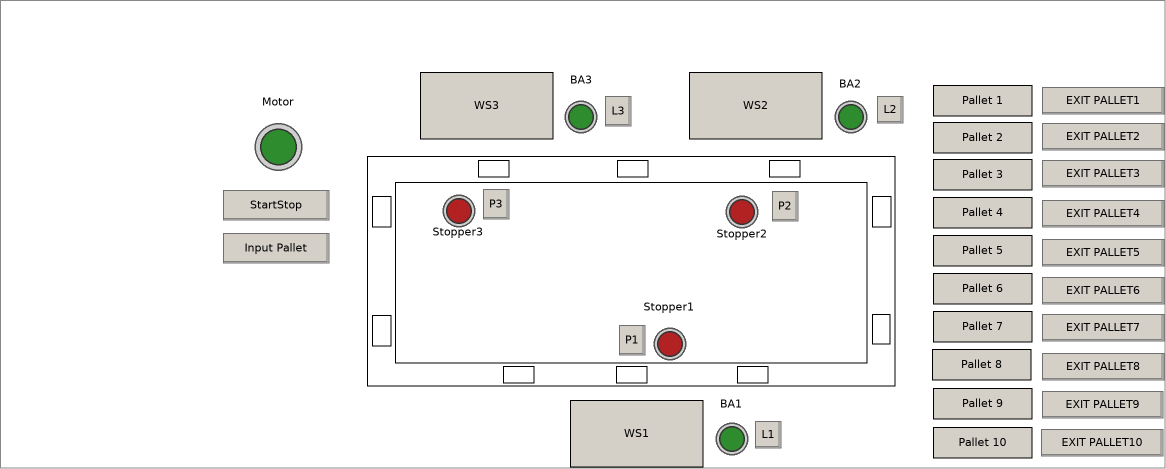
VISUALIZATION Visualization  // 1166x469
    RoundedRectangle (367,156 528x230)
    RoundedRectangle (395,182 472x181)
    Rectangle (570,400 133x67), "WS1", colour toggle: MAIN.T1.Q
    Rectangle (420,72 133x67), "WS3", colour toggle: MAIN.T3.Q
    Rectangle (689,72 133x67), "WS2", colour toggle: MAIN.T2.Q
    Button (755,421 26x27), "L1", text variable: MAIN.L1, colour toggle: MAIN.L1
        toggle MAIN.L1
    Button (605,96 26x30), "L3", text variable: MAIN.L3, colour toggle: MAIN.L3
        toggle MAIN.L3
    Button (483,189 26x30), "P3"
        tap MAIN.P3
    Button (772,191 26x30), "P2"
        tap MAIN.P2
    Button (619,325 26x30), "P1"
        tap MAIN.P1
    Lamp1 (832,94 38x46), tooltip "BA2", variable: MAIN.BA2, style: Lamp-Lamp1-Green
    Label (775,69 150x30), "BA2"
    Lamp1 (562,94 38x46), variable: MAIN.BA3, style: Lamp-Lamp1-Green
    Lamp1 (713,416 38x46), variable: MAIN.BA1, style: Lamp-Lamp1-Green
    Label (506,63 150x34), "BA3"
    Label (656,389 150x30), "BA1"
    Lamp1 (723,189 38x46), variable: MAIN.S2, style: Lamp-Lamp1-Red
    Lamp1 (440,188 38x46), variable: MAIN.S3, style: Lamp-Lamp1-Red
    Lamp1 (651,321 38x46), variable: MAIN.S1, style: Lamp-Lamp1-Red
    Label (594,292 150x30), "Stopper1"
    Label (383,217 150x30), "Stopper3"
    Label (667,219 150x30), "Stopper2"
    Rectangle (503,366 31x17)
    Lamp1 (251,115 55x64), variable: MAIN.MOTOR, style: Lamp-Lamp1-Green
    Label (203,87 150x30), "Motor"
    Button (223,190 106x30), "StartStop"
        toggle MAIN.StartStop
    Button (223,233 106x30), "Input Pallet"
        tap MAIN.INPUT_PALLET_Pressed
    Button (877,96 26x27), "L2", text variable: MAIN.L2, colour toggle: MAIN.L2
        toggle MAIN.L2
    Rectangle (933,85 99x31), "Pallet 1", colour toggle: MAIN.PALLETV[2].WS1
    Rectangle (372,315 19x31)
    Rectangle (617,160 31x17)
    Rectangle (769,160 31x17), invisible if: MAIN.L2
    Rectangle (478,160 31x17), invisible if: MAIN.L3
    Rectangle (737,366 31x17)
    Rectangle (616,366 31x17), invisible if: MAIN.L1
    Rectangle (872,314 18x30)
    Rectangle (872,196 19x31)
    Rectangle (372,196 19x31)
    Rectangle (933,122 99x31), "Pallet 2", colour toggle: MAIN.PALLETV[3].WS1
    Rectangle (933,159 99x31), "Pallet 3", colour toggle: MAIN.PALLETV[4].WS1
    Rectangle (933,197 99x31), "Pallet 4", colour toggle: MAIN.PALLETV[5].WS1
    Rectangle (933,235 99x31), "Pallet 5", colour toggle: MAIN.PALLETV[6].WS1
    Rectangle (933,273 99x31), "Pallet 6", colour toggle: MAIN.PALLETV[7].WS1
    Rectangle (933,311 99x31), "Pallet 7", colour toggle: MAIN.PALLETV[8].WS1
    Rectangle (932,349 99x31), "Pallet 8", colour toggle: MAIN.PALLETV[9].WS1
    Rectangle (933,388 99x31), "Pallet 9", colour toggle: MAIN.PALLETV[10].WS1
    Rectangle (933,427 99x31), "Pallet 10", colour toggle: MAIN.PALLETV[11].WS1
    Button (1041,429 122x27), "EXIT PALLET10"
        tap MAIN.RESET_OUTV11
    Button (1042,160 122x27), "EXIT PALLET3"
        tap MAIN.RESET_OUTV4
    Button (1042,200 122x27), "EXIT PALLET4"
        tap MAIN.RESET_OUTV5
    Button (1042,239 122x27), "EXIT PALLET5"
        tap MAIN.RESET_OUTV6
    Button (1042,277 122x27), "EXIT PALLET6"
        tap MAIN.RESET_OUTV7
    Button (1042,314 122x27), "EXIT PALLET7"
        tap MAIN.RESET_OUTV8
    Button (1042,353 122x27), "EXIT PALLET8"
        tap MAIN.RESET_OUTV9
    Button (1042,391 121x27), "EXIT PALLET9"
        tap MAIN.RESET_OUTV10
    Button (1042,123 122x27), "EXIT PALLET2"
        tap MAIN.RESET_OUTV3
    Button (1042,87 122x27), "EXIT PALLET1"
        tap MAIN.RESET_OUTV2
END_VISUALIZATION

(* stored: Version 1.1.0.1, ProductVersion 3.1.4020.12
   Visu Visualization: Id {aba1789d-4405-4121-8f5b-68c61a8109f6} *)
